FUNCTION_BLOCK ENCODERPULSEtoANGLE
VAR_INPUT
	A :BOOL;
	B:BOOL;
	Pulsos:DINT:=1600;
	b_calibrado: BOOL;
	angulo_calibrado : REAL;
END_VAR
VAR_OUTPUT
	acum : DINT:=0;
	angle :REAL;
	estado : INT;
END_VAR
VAR
	delta_angulo : REAL;
END_VAR

//determinar delta angulo
delta_angulo:=2*GVL.pi/pulsos;

//ACUM
CASE estado OF
	0: //INIT
	IF(A AND NOT(B)) THEN
		estado:=1;
		ELSE IF A AND B THEN
			estado:=2;
			ELSE IF B AND NOT(A) THEN
				estado:=3;
				ELSE IF NOT(B)AND NOT(A) THEN
					estado:=4;
				END_IF
			END_IF
			
		END_IF
	END_IF
	estado:=1;
	1:
	IF B THEN
		estado:=2;
		acum:=acum+1;
		angle:=angle + delta_angulo;
		ELSE IF NOT(A) THEN
			estado:=4;
			acum:=acum-1;
			angle:=angle - delta_angulo;
		END_IF
	END_IF
	2:
	IF NOT(A) THEN
		estado:=3;
		acum:=acum+1;
		angle:=angle + delta_angulo;
		ELSE IF NOT(B) THEN
			estado:=1;
			acum:=acum-1;
			angle:=angle - delta_angulo;
		END_IF
	END_IF
	3:
	IF NOT(B) THEN
		estado:=4;
		acum:=acum+1;
		angle:=angle + delta_angulo;
		ELSE IF A THEN
			estado:=2;
			acum:=acum-1;
			angle:=angle - delta_angulo;
		END_IF
	END_IF
	4:
	IF A THEN
		estado:=1;
		acum:=acum+1;
		angle:=angle + delta_angulo;
		ELSE IF B THEN
			estado:=3;
			acum:=acum-1;
			angle:=angle - delta_angulo;
		END_IF
	END_IF
	
END_CASE

//calibración
IF b_calibrado THEN
	acum:=0;
	angle:=angulo_calibrado;	
END_IF

END_FUNCTION_BLOCK

(* stored: Version 1.1.0.1, ProductVersion 3.1.4024.4
   POU ENCODERPULSEtoANGLE: Id {e4835318-288f-4071-898a-39471c291f8c}, SpecialFunc None *)
